TEXTLIST TextList_Config_EFFLUVAGE
  0 = 'Effluvage' | FR: 'EFFLUVAGE' | EN: 'GLOW DISCHARGE'
  1 = 'PRM_Tp_Vent' | FR: 'Température max. pour ventilation enceinte' | EN: 'Max. temperature for chamber venting'
  2 = 'PRM_Max_Temp' | FR: 'Consigne température max.' | EN: 'Max. temperature setpoint'
  3 = 'CONF_Pmax' | FR: 'Puissance max.' | EN: 'Max. setpoint'
  4 = 'P' | FR: 'Gain' | EN: 'Amplification factor'
  5 = 'Ti' | FR: "Temps d'action intégrale" | EN: 'Integral action time'
  6 = 'Td' | FR: "Temps d'action dérivée" | EN: 'Derivative action time'
  7 = 'Ta' | FR: "Temps d'amortissement" | EN: 'Damping time'
  8 = 'Tc Ctrl' | FR: 'Seuil de courant de détéction du plasma' | EN: 'Plasma current detection threshold'
  9 = 'Tc Disp' | FR: 'Seuil de tension de détéction du plasma' | EN: 'Plasma voltage detection threshold'
  10 = 'Alimentation' | FR: 'ALIMENTATION' | EN: 'POWER SUPPLY'
  11 = 'alm surv delay' | FR: 'Temps de surveillance avant alarme' | EN: 'Delay before alarm'
  12 = 'alm surv offset' | FR: 'Offset de surveillance avant alarme' | EN: 'Offset before alarm'
  13 = 'dft surv delay' | FR: 'Temps de surveillance avant défaut' | EN: 'Delay before fault'
  14 = 'dft surv offset' | FR: 'Offset de surveillance avant défaut' | EN: 'Offset before fault'
   = ''
END_TEXTLIST

(* stored: Version 1.1.0.1, ProductVersion 3.1.4024.10
   TextList TextList_Config_EFFLUVAGE: Id {86a2f90f-6cdf-4674-bbf0-a482513eb7d3} *)
